Omron CX-Programmer project НовыйПроект (CX-Programmer 9.73)

# PLC НовыйПЛК1: CP1L-E EL

## Program НоваяЗадача1 (cyclic task 0)
Local symbols
Accel_SM D10 UINT  ; Скорость разгона (шагового мотора)
Decel_SM D11 UINT  ; Скорость торможения (шагового мотора)
Hold_off 100.02 BOOL
Init_Freq D16 UDINT  ; Начальное значение частоты (шаговый мотор)
Level_led 0.02 BOOL
Power_key 100.03 BOOL
Power_led 0.01 BOOL  ; индикатор включенного состояния
Target_Freq D12 UDINT  ; Целевая частота вращения (шагового мотора)
Target_Step D14 UDINT  ; Целевое кол-во шаговых импульсов (шагового мотора)
back_spin W0.01 BOOL
current_angle W4 INT
fins_byte_out W2 INT
luft_value D18 UDINT  ; количество импульсов на компенсацию люфта
r_sw 0.00 BOOL  ; геркон
some_out 100.02 BOOL  ; просто выход
state W1 INT
step0 W0.03 BOOL
step1 W0.01 BOOL
step2 W0.02 BOOL

### Section инициализация

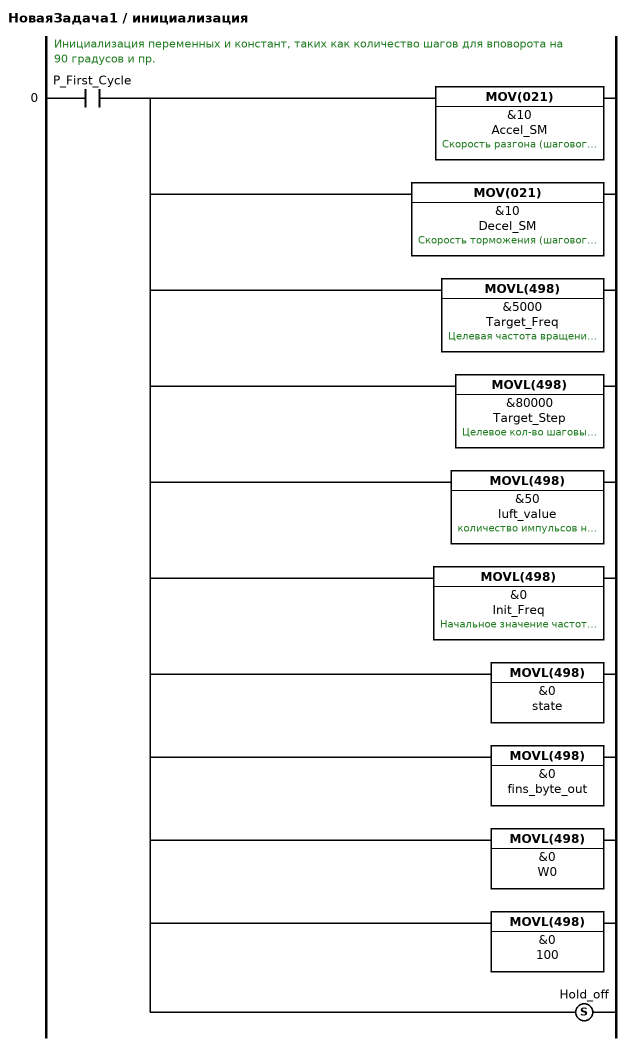
; rung 0: Инициализация переменных и констант, таких как количество шагов для вповорота на 90 градусов и пр.
LD P_First_Cycle
MOV(021) &10 Accel_SM  ; Скорость разгона (шагового мотора)
MOV(021) &10 Decel_SM  ; Скорость торможения (шагового мотора)
MOVL(498) &5000 Target_Freq  ; Целевая частота вращения (шагового мотора)
MOVL(498) &80000 Target_Step  ; Целевое кол-во шаговых импульсов (шагового мотора)
MOVL(498) &50 luft_value  ; количество импульсов на компенсацию люфта
MOVL(498) &0 Init_Freq  ; Начальное значение частоты (шаговый мотор)
MOVL(498) &0 state
MOVL(498) &0 fins_byte_out
MOVL(498) &0 W0
MOVL(498) &0 100
SET Hold_off

### Section установка_в_начало_по_геркону

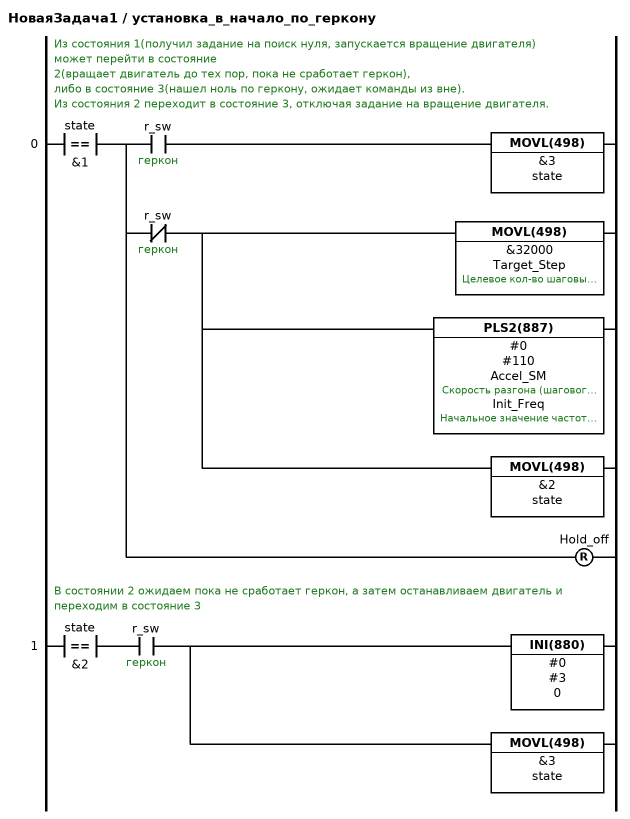
; rung 0: Из состояния 1(получил задание на поиск нуля, запускается вращение двигателя) может перейти в состояние / 2(вращает двигатель до тех пор, пока не сработает геркон), / либо в состояние 3(нашел ноль по геркону, ожидает команды из вне). / Из состояния 2 переходит в состояние 3, отключая задание на вращение двигателя.
LD=(300) state &1
OUT TR0
AND r_sw  ; геркон
MOVL(498) &3 state
LD TR0
ANDNOT r_sw  ; геркон
MOVL(498) &32000 Target_Step  ; Целевое кол-во шаговых импульсов (шагового мотора)
PLS2(887) #0 #110 Accel_SM Init_Freq  ; Скорость разгона (шагового мотора), Начальное значение частоты (шаговый мотор)
MOVL(498) &2 state
LD TR0
RSET Hold_off
; rung 1: В состоянии 2 ожидаем пока не сработает геркон, а затем останавливаем двигатель и переходим в состояние 3
LD=(300) state &2
AND r_sw  ; геркон
INI(880) #0 #3 0
MOVL(498) &3 state

### Section включение_прибора

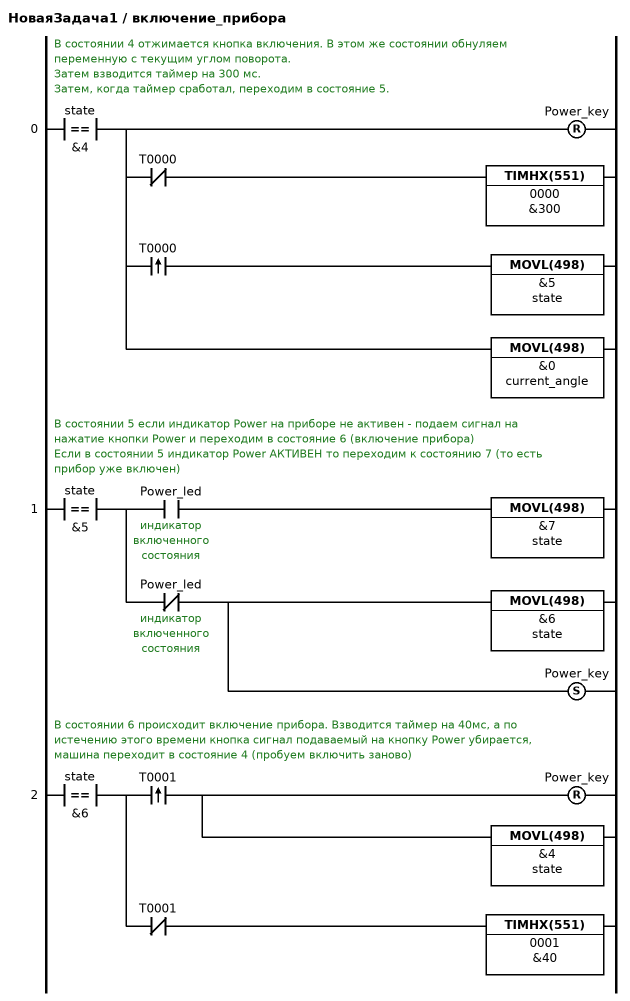
; rung 0: В состоянии 4 отжимается кнопка включения. В этом же состоянии обнуляем переменную с текущим углом поворота. / Затем взводится таймер на 300 мс. / Затем, когда таймер сработал, переходим в состояние 5.
LD=(300) state &4
OUT TR0
RSET Power_key
ANDNOT T0000
TIMHX(551) 0000 &300
LD TR0
@AND T0000
MOVL(498) &5 state
LD TR0
MOVL(498) &0 current_angle
; rung 1: В состоянии 5 если индикатор Power на приборе не активен - подаем сигнал на нажатие кнопки Power и переходим в состояние 6 (включение прибора) / Если в состоянии 5 индикатор Power АКТИВЕН то переходим к состоянию 7 (то есть прибор уже включен)
LD=(300) state &5
OUT TR0
AND Power_led  ; индикатор включенного состояния
MOVL(498) &7 state
LD TR0
ANDNOT Power_led  ; индикатор включенного состояния
MOVL(498) &6 state
SET Power_key
; rung 2: В состоянии 6 происходит включение прибора. Взводится таймер на 40мс, а по истечению этого времени кнопка сигнал подаваемый на кнопку Power убирается, машина переходит в состояние 4 (пробуем включить заново)
LD=(300) state &6
OUT TR0
@AND T0001
RSET Power_key
MOVL(498) &4 state
LD TR0
ANDNOT T0001
TIMHX(551) 0001 &40

### Section ожидание_стабилизации_1

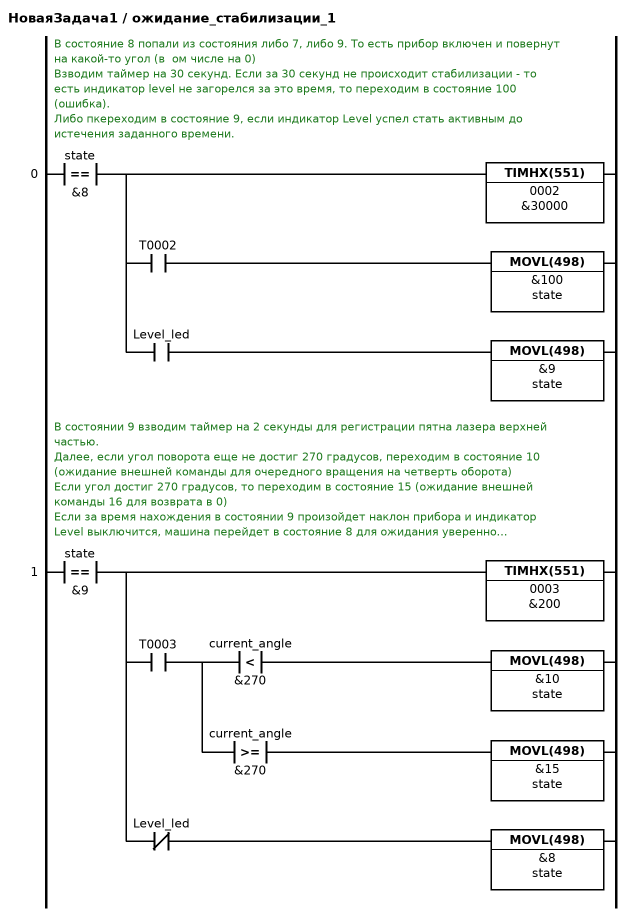
; rung 0: В состояние 8 попали из состояния либо 7, либо 9. То есть прибор включен и повернут на какой-то угол (в  ом числе на 0) / Взводим таймер на 30 секунд. Если за 30 секунд не происходит стабилизации - то есть индикатор level не загорелся за это время, то переходим в состояние 100 (ошибка). / Либо пкереходим в состояние 9, если индикатор Level успел стать активным до истечения заданного времени.
LD=(300) state &8
OUT TR0
TIMHX(551) 0002 &30000
AND T0002
MOVL(498) &100 state
LD TR0
AND Level_led
MOVL(498) &9 state
; rung 1: В состоянии 9 взводим таймер на 2 секунды для регистрации пятна лазера верхней частью. / Далее, если угол поворота еще не достиг 270 градусов, переходим в состояние 10 (ожидание внешней команды для очередного вращения на четверть оборота) / Если угол достиг 270 градусов, то переходим в состояние 15 (ожидание внешней команды 16 для возврата в 0) / Если за время нахождения в состоянии 9 произойдет наклон прибора и индикатор Level выключится, машина перейдет в состояние 8 для ожидания уверенной стабилизации.
LD=(300) state &9
OUT TR0
TIMHX(551) 0003 &200
AND T0003
OUT TR1
AND<(310) current_angle &270
MOVL(498) &10 state
LD TR1
AND>=(325) current_angle &270
MOVL(498) &15 state
LD TR0
ANDNOT Level_led
MOVL(498) &8 state

### Section поворот_1

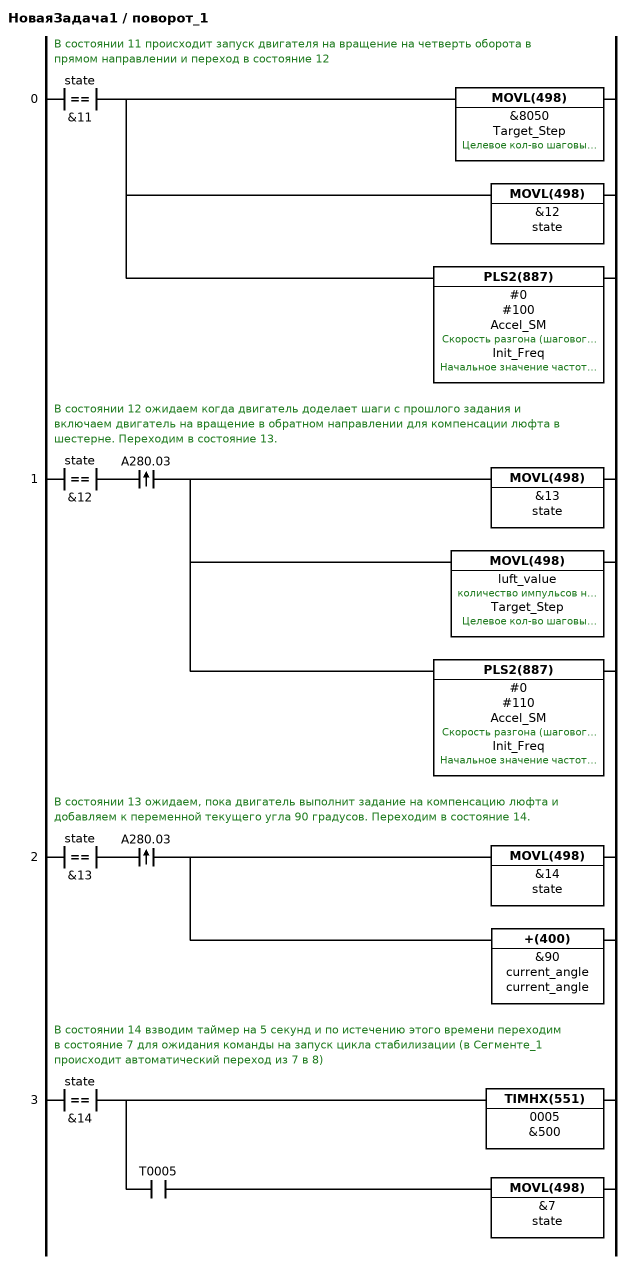
; rung 0: В состоянии 11 происходит запуск двигателя на вращение на четверть оборота в прямом направлении и переход в состояние 12
LD=(300) state &11
MOVL(498) &8050 Target_Step  ; Целевое кол-во шаговых импульсов (шагового мотора)
MOVL(498) &12 state
PLS2(887) #0 #100 Accel_SM Init_Freq  ; Скорость разгона (шагового мотора), Начальное значение частоты (шаговый мотор)
; rung 1: В состоянии 12 ожидаем когда двигатель доделает шаги с прошлого задания и включаем двигатель на вращение в обратном направлении для компенсации люфта в шестерне. Переходим в состояние 13.
LD=(300) state &12
@AND A280.03
MOVL(498) &13 state
MOVL(498) luft_value Target_Step  ; количество импульсов на компенсацию люфта, Целевое кол-во шаговых импульсов (шагового мотора)
PLS2(887) #0 #110 Accel_SM Init_Freq  ; Скорость разгона (шагового мотора), Начальное значение частоты (шаговый мотор)
; rung 2: В состоянии 13 ожидаем, пока двигатель выполнит задание на компенсацию люфта и добавляем к переменной текущего угла 90 градусов. Переходим в состояние 14.
LD=(300) state &13
@AND A280.03
MOVL(498) &14 state
+(400) &90 current_angle current_angle
; rung 3: В состоянии 14 взводим таймер на 5 секунд и по истечению этого времени переходим в состояние 7 для ожидания команды на запуск цикла стабилизации (в Сегменте_1 происходит автоматический переход из 7 в 8)
LD=(300) state &14
TIMHX(551) 0005 &500
AND T0005
MOVL(498) &7 state

### Section возврат_в_ноль

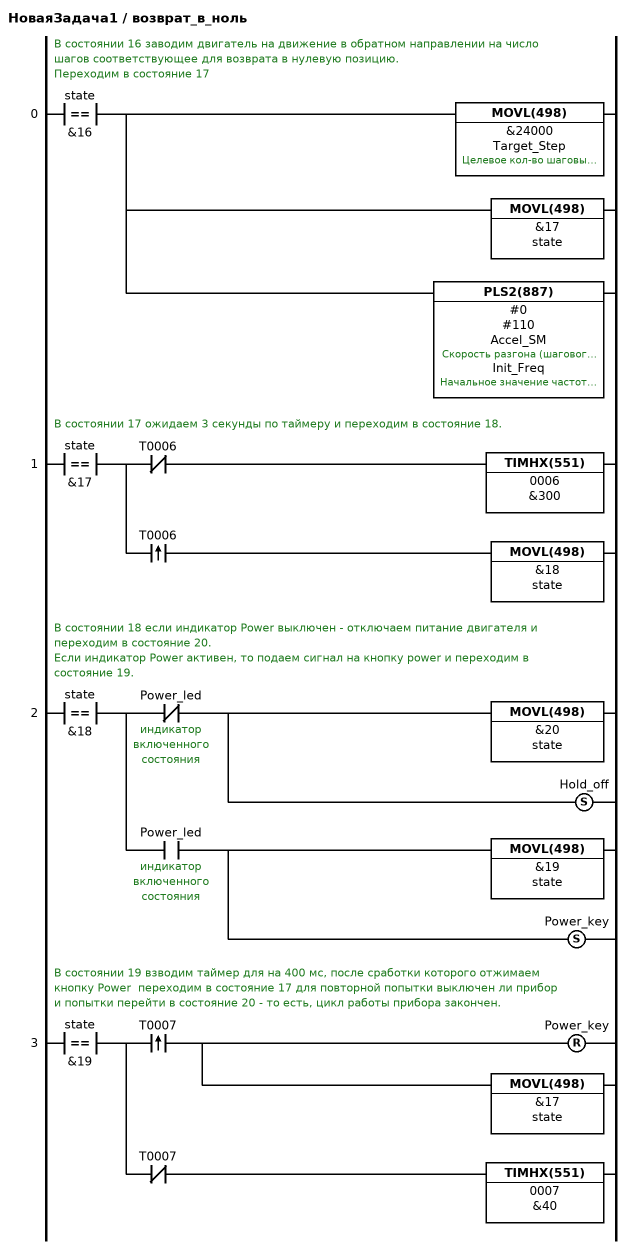
; rung 0: В состоянии 16 заводим двигатель на движение в обратном направлении на число шагов соответствующее для возврата в нулевую позицию. / Переходим в состояние 17
LD=(300) state &16
MOVL(498) &24000 Target_Step  ; Целевое кол-во шаговых импульсов (шагового мотора)
MOVL(498) &17 state
PLS2(887) #0 #110 Accel_SM Init_Freq  ; Скорость разгона (шагового мотора), Начальное значение частоты (шаговый мотор)
; rung 1: В состоянии 17 ожидаем 3 секунды по таймеру и переходим в состояние 18.
LD=(300) state &17
OUT TR0
ANDNOT T0006
TIMHX(551) 0006 &300
LD TR0
@AND T0006
MOVL(498) &18 state
; rung 2: В состоянии 18 если индикатор Power выключен - отключаем питание двигателя и переходим в состояние 20. / Если индикатор Power активен, то подаем сигнал на кнопку power и переходим в состояние 19.
LD=(300) state &18
OUT TR0
ANDNOT Power_led  ; индикатор включенного состояния
MOVL(498) &20 state
SET Hold_off
LD TR0
AND Power_led  ; индикатор включенного состояния
MOVL(498) &19 state
SET Power_key
; rung 3: В состоянии 19 взводим таймер для на 400 мс, после сработки которого отжимаем кнопку Power  переходим в состояние 17 для повторной попытки выключен ли прибор и попытки перейти в состояние 20 - то есть, цикл работы прибора закончен.
LD=(300) state &19
OUT TR0
@AND T0007
RSET Power_key
MOVL(498) &17 state
LD TR0
ANDNOT T0007
TIMHX(551) 0007 &40

### Section Сегмент1

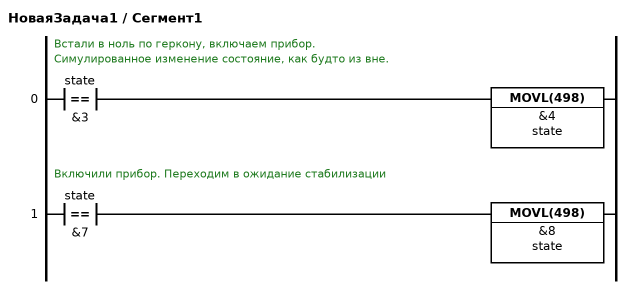
; rung 0: Встали в ноль по геркону, включаем прибор. / Симулированное изменение состояние, как будто из вне.
LD=(300) state &3
MOVL(498) &4 state
; rung 1: Включили прибор. Переходим в ожидание стабилизации
LD=(300) state &7
MOVL(498) &8 state
; rung 2
END(001)